// Mitsubishi GX Works2 project: AD input 0-10V Python   PLC: FX3U/FX3UC

PROGRAM MAIN
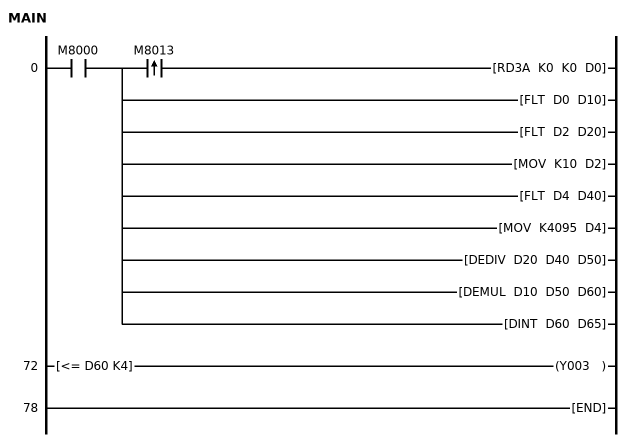
0     LD      M8000
      MPS
      ANDP    M8013
      RD3A    K0 K0 D0
      MPP
      FLT     D0 D10
      FLT     D2 D20
      MOV     K10 D2
      FLT     D4 D40
      MOV     K4095 D4
      DEDIV   D20 D40 D50
      DEMUL   D10 D50 D60
      DINT    D60 D65
72    LD<=    D60 K4
      OUT     Y003
78    END
END_PROGRAM
